// LS Electric XG5000 project: fdas
// PLC NewPLC
// module base 0 slot 0: 입출력 모듈:XBC-DR32H (DC 24V 입력, 릴레이 출력 32점)
// module base 0 slot 1: 위치결정 모듈:XBF-PD02A (위치결정 펄스(LD)출력형, 2축)
// module base 0 slot 2: 출력 모듈:XBE-TN/TP16A (트랜지스터 출력, 16점 (싱크출력/소스출력))

PROGRAM NewProgram (task: 스캔 프로그램)

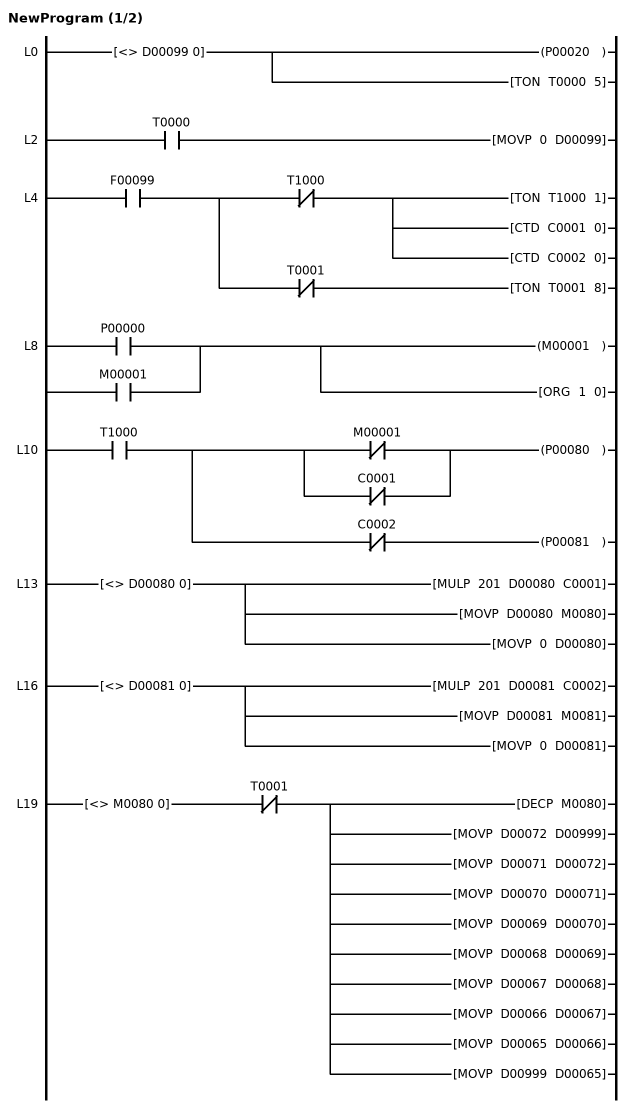
; L0
LOAD<>    D00099 0
OUT       P00020
TON       T0000 5
; L2
LOAD      T0000
MOVP      0 D00099
; L4
LOAD      F00099
MPUSH
AND NOT   T1000
TON       T1000 1
CTD       C0001 0
CTD       C0002 0
MPOP
AND NOT   T0001
TON       T0001 8
; L8
LOAD      P00000
OR        M00001
OUT       M00001
ORG       1 0
; L10
LOAD      T1000
MPUSH
LOAD NOT  M00001
OR NOT    C0001
AND LOAD
OUT       P00080
MPOP
AND NOT   C0002
OUT       P00081
; L13
LOAD<>    D00080 0
MULP      201 D00080 C0001
MOVP      D00080 M0080
MOVP      0 D00080
; L16
LOAD<>    D00081 0
MULP      201 D00081 C0002
MOVP      D00081 M0081
MOVP      0 D00081
; L19
LOAD<>    M0080 0
AND NOT   T0001
DECP      M0080
MOVP      D00072 D00999
MOVP      D00071 D00072
MOVP      D00070 D00071
MOVP      D00069 D00070
MOVP      D00068 D00069
MOVP      D00067 D00068
MOVP      D00066 D00067
MOVP      D00065 D00066
MOVP      D00999 D00065

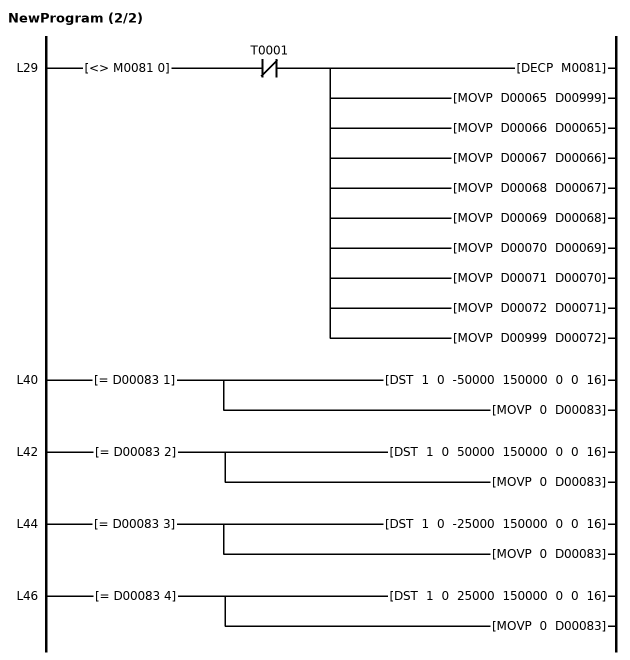
; L29
LOAD<>    M0081 0
AND NOT   T0001
DECP      M0081
MOVP      D00065 D00999
MOVP      D00066 D00065
MOVP      D00067 D00066
MOVP      D00068 D00067
MOVP      D00069 D00068
MOVP      D00070 D00069
MOVP      D00071 D00070
MOVP      D00072 D00071
MOVP      D00999 D00072
; L40
LOAD=     D00083 1
DST       1 0 -50000 150000 0 0 16
MOVP      0 D00083
; L42
LOAD=     D00083 2
DST       1 0 50000 150000 0 0 16
MOVP      0 D00083
; L44
LOAD=     D00083 3
DST       1 0 -25000 150000 0 0 16
MOVP      0 D00083
; L46
LOAD=     D00083 4
DST       1 0 25000 150000 0 0 16
MOVP      0 D00083